# EPICS IOC start-up script: commonIocsh/iocsh/linStatProc.iocsh
#--################################################################################################
#--############### START of linStatProc.iocsh #####################################################
#-- IOC     : Record name prefix
#-- LINSTAT : linStat module install top (db under $(LINSTAT)/db)
#--################################################################################################
#--#
#--# This IOC's process statistics: memory, file descriptors, threads, CA client count, records.
#--# Load before iocInit. Loaded by default from the global linStat.iocsh.
#--#
#--# Do not load together with iocStatsAdmin.iocsh for the same IOC: both create records of the
#--# same names, and the second load fails.
#--#
#-
dbLoadRecords("$(LINSTAT)/db/linStatProc.db", "IOC=$(IOC)")
#-
#--############### END of linStatProc.iocsh #######################################################
#--################################################################################################
